// TIA Portal V18 export
FUNCTION_BLOCK "encoder"   // FB15, FBD
{ S7_Optimized_Access := 'TRUE' }
VERSION : 0.1
// stored: AutoNumber true, IsIECCheckEnabled false, IsRetainMemResEnabled false, MemoryReserve 100, SetENOAutomatically false, UDAEnableTagReadback false
   VAR_INPUT
      isMultiturn : Bool;
      pos_lim_fwd : Real;
      pos_lim_rev : Real;
      ENC : Real;
      par_calpos_predef : Real;
      xPredefCal : Bool;
   END_VAR
   VAR_OUTPUT
      POS : Real;
      calibrated : Bool;
      saved_fwd : Real;
      saved_rev : Real;
      ER_set : Bool;
      ER_w : WString;
   END_VAR
   VAR_IN_OUT
      RET_DATA : "typePOSMEMcalib";
      target_pos : Real;
   END_VAR
   VAR
      not_first_scan : Bool;
      xPredefCal_filtered : Bool;
      tr_predef : R_TRIG;
      tr_fwd : R_TRIG;
      tr_rev : R_TRIG;
      ton_filter { S7_SetPoint := 'True'} : TON_TIME;
   END_VAR
   VAR_TEMP
      btn_calib_now_predef : Bool;
      btn_calib_now_fwd : Bool;
      btn_calib_now_rev : Bool;
      length_rev_fwd : Real;
   END_VAR
BEGIN

REGION Network 1
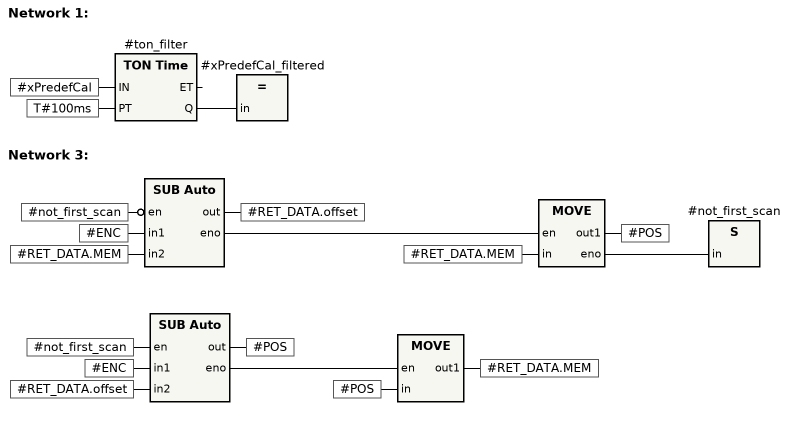
   #ton_filter(IN := #xPredefCal, PT := T#100ms);   // TON
   #xPredefCal_filtered := #ton_filter.Q;
END_REGION

REGION Network 2 (SCL)
   IF #isMultiturn THEN
       IF NOT #RET_DATA.calibrated THEN
           #RET_DATA.calibrated := true;
       END_IF;
       IF #pos_lim_fwd > #pos_lim_rev THEN
           #ER_set := false;
           #ER_w := WString#'';
           #length_rev_fwd := #pos_lim_fwd - #pos_lim_rev;
           IF #POS >= #pos_lim_fwd THEN


               #RET_DATA.offset := #RET_DATA.offset + #length_rev_fwd;
           END_IF;
           IF #POS < #pos_lim_rev THEN
               #RET_DATA.offset := #RET_DATA.offset - #length_rev_fwd;
           END_IF;



           IF #target_pos >= #pos_lim_fwd THEN
               #target_pos := #target_pos - #length_rev_fwd;
           END_IF;
           IF #target_pos < #pos_lim_rev THEN
               #target_pos := #target_pos + #length_rev_fwd;
           END_IF;
       ELSE
           #ER_set := true;
           #ER_w := WString#'enc_fwd_lt_rev';
       END_IF;
   END_IF;
END_REGION

REGION Network 3
   IF NOT #not_first_scan THEN
       #RET_DATA.offset := #ENC - #RET_DATA.MEM;
       #POS := #RET_DATA.MEM;
       #not_first_scan := TRUE;
   END_IF;
   IF #not_first_scan THEN
       #POS := #ENC - #RET_DATA.offset;
       #RET_DATA.MEM := #POS;
   END_IF;
END_REGION

REGION Network 4 (SCL)
   #tr_predef(CLK := #xPredefCal_filtered);

   #btn_calib_now_predef := #tr_predef.Q;

   IF #btn_calib_now_predef THEN
       #RET_DATA.offset := #ENC - #par_calpos_predef;
       #RET_DATA.calibrated := true;
   END_IF;

   #calibrated := #RET_DATA.calibrated;
END_REGION
END_FUNCTION_BLOCK
